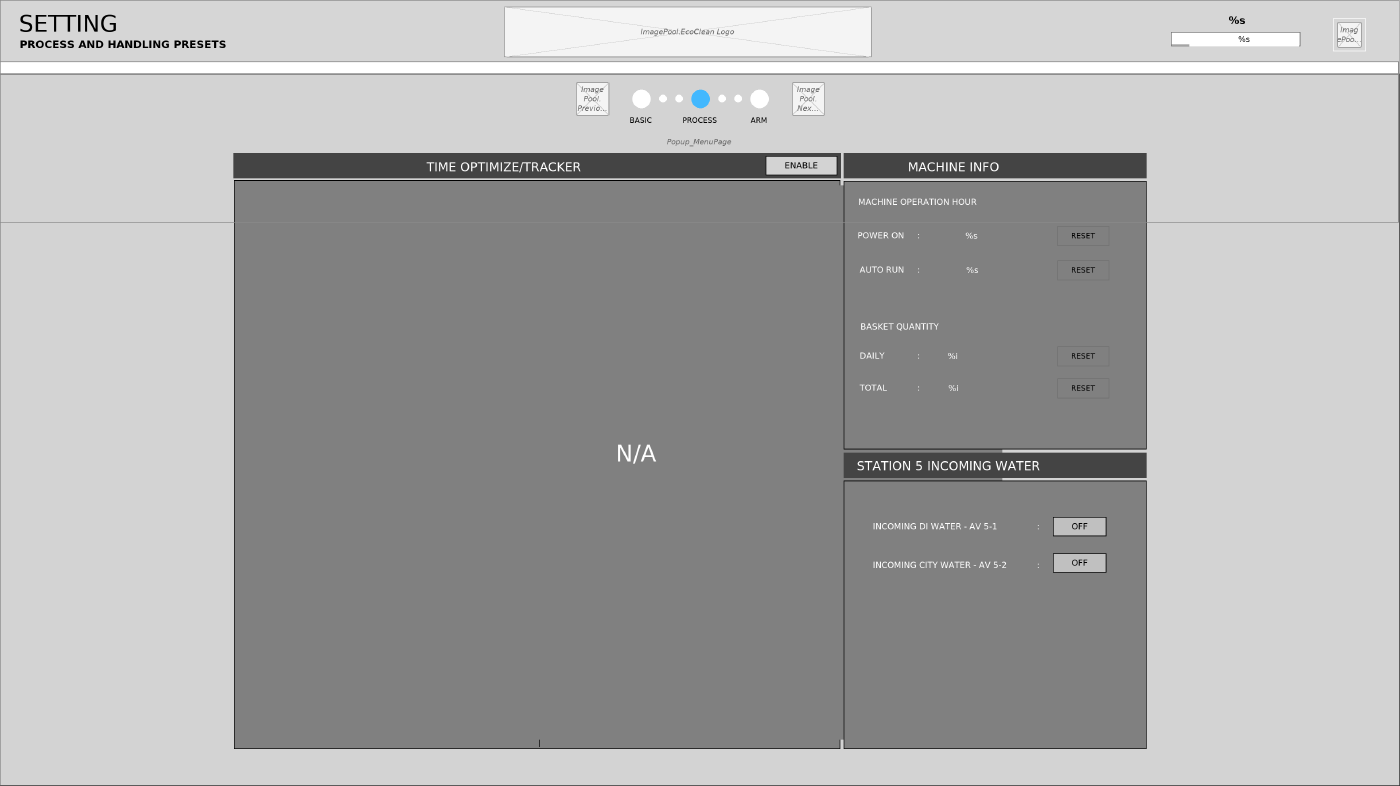
VISUALIZATION SettingProcess_Page  // 1920x1078
    Rectangle (0,101 1920x977)
    Rectangle (321,247 831x780)
    Rectangle (0,63 1920x26)
        p3528305787: HMI_Ctrl.ANIMATION3
    Rectangle (0,0 1919x85)
    Label (23,6 267x53), "SETTING"
    Label (24,49 320x24), "PROCESS AND HANDLING PRESETS"
    Group (1828,25 45x45)
        OnMouseClick: toggle HMI_Ctrl.MenuButton
        RoundedRectangle (0,0 45x45), colour toggle: HMI_Ctrl.MenuButton
        Image (6,5 33x35), image: ImagePool.Menu Button
    Ellipse (867,123 25x25)
    Ellipse (948,123 25x25)
    Ellipse (904,130 10x10)
    Ellipse (926,130 10x10)
    Ellipse (985,130 10x10)
    Ellipse (1007,130 10x10)
    Ellipse (1029,123 25x25)
    Label (847,153 64x24), "BASIC"
    Label (928,153 64x24), "PROCESS"
    Label (1009,153 64x24), "ARM"
    Image (1086,113 45x45), image: ImagePool.Next Button
        OnMouseClick: change screen: SettingArm_Page
    Image (790,113 45x45), image: ImagePool.Previous Button
        OnMouseClick: change screen: Setting_Page
    Rectangle (320,210 833x34)
    Label (582,217 283x24), "TIME OPTIMIZE/TRACKER"
    RoundedRectangle (491,308 30x30), colour toggle: ARbProductRecipeTimeBlockAvailable[1]
    RoundedRectangle (491,378 30x30), colour toggle: ARbProductRecipeTimeBlockAvailable[2]
    RoundedRectangle (491,446 30x30), colour toggle: ARbProductRecipeTimeBlockAvailable[3]
    RoundedRectangle (491,523 30x30), colour toggle: ARbProductRecipeTimeBlockAvailable[4]
    RoundedRectangle (491,598 30x30), colour toggle: ARbProductRecipeTimeBlockAvailable[5]
    RoundedRectangle (491,678 30x30), colour toggle: ARbProductRecipeTimeBlockAvailable[6]
    RoundedRectangle (491,758 30x30), colour toggle: ARbProductRecipeTimeBlockAvailable[7]
    RoundedRectangle (491,829 30x30), colour toggle: ARbProductRecipeTimeBlockAvailable[8]
    RoundedRectangle (491,898 30x30), colour toggle: ARbProductRecipeTimeBlockAvailable[9]
    Label (484,260 103x25), "ENABLE"
    RoundedRectangle (491,968 30x30), colour toggle: ARbProductRecipeTimeBlockAvailable[10]
    Label (385,307 37x24), "1"
    Label (385,377 37x24), "2"
    Label (385,445 37x24), "3"
    Label (385,522 37x24), "4"
    Label (385,597 37x24), "5"
    Label (385,677 37x24), "6"
    Label (385,757 37x24), "7"
    Label (385,828 37x24), "8"
    Label (385,897 37x24), "9"
    Label (380,967 37x24), "10"
    Label (360,248 113x46), "RECIPE NO"
    RoundedRectangle (594,306 90x40), "RESET", input disabled if: bMainOnOff
        tap bTrackerReset[1]
    RoundedRectangle (594,376 90x40), "RESET", input disabled if: bMainOnOff
        tap bTrackerReset[2]
    RoundedRectangle (594,444 90x40), "RESET", input disabled if: bMainOnOff
        tap bTrackerReset[3]
    RoundedRectangle (594,521 90x40), "RESET", input disabled if: bMainOnOff
        tap bTrackerReset[4]
    RoundedRectangle (594,596 90x40), "RESET", input disabled if: bMainOnOff
        tap bTrackerReset[5]
    RoundedRectangle (594,676 90x40), "RESET", input disabled if: bMainOnOff
        tap bTrackerReset[6]
    RoundedRectangle (594,756 90x40), "RESET", input disabled if: bMainOnOff
        tap bTrackerReset[7]
    RoundedRectangle (594,827 90x40), "RESET", input disabled if: bMainOnOff
        tap bTrackerReset[8]
    RoundedRectangle (594,896 90x40), "RESET", input disabled if: bMainOnOff
        tap bTrackerReset[9]
    RoundedRectangle (594,966 90x40), "RESET", input disabled if: bMainOnOff
        tap bTrackerReset[10]
    RoundedRectangle (906,308 30x30), colour toggle: ARbProductRecipeTimeBlockAvailable[11]
    RoundedRectangle (906,378 30x30), colour toggle: ARbProductRecipeTimeBlockAvailable[12]
    RoundedRectangle (906,446 30x30), colour toggle: ARbProductRecipeTimeBlockAvailable[13]
    RoundedRectangle (906,523 30x30), colour toggle: ARbProductRecipeTimeBlockAvailable[14]
    RoundedRectangle (906,598 30x30), colour toggle: ARbProductRecipeTimeBlockAvailable[15]
    RoundedRectangle (906,678 30x30), colour toggle: ARbProductRecipeTimeBlockAvailable[16]
    RoundedRectangle (906,758 30x30), colour toggle: ARbProductRecipeTimeBlockAvailable[17]
    RoundedRectangle (906,829 30x30), colour toggle: ARbProductRecipeTimeBlockAvailable[18]
    RoundedRectangle (906,898 30x30), colour toggle: ARbProductRecipeTimeBlockAvailable[19]
    Label (894,258 103x25), "ENABLE"
    RoundedRectangle (906,968 30x30), colour toggle: ARbProductRecipeTimeBlockAvailable[20]
    Label (803,309 37x24), "11"
    Label (803,379 37x24), "12"
    Label (803,447 37x24), "13"
    Label (803,524 37x24), "14"
    Label (803,599 37x24), "15"
    Label (803,679 37x24), "16"
    Label (803,759 37x24), "17"
    Label (803,830 37x24), "18"
    Label (803,899 37x24), "19"
    Label (802,969 37x24), "20"
    RoundedRectangle (1007,306 90x40), "RESET", input disabled if: bMainOnOff
        tap bTrackerReset[11]
    RoundedRectangle (1007,376 90x40), "RESET", input disabled if: bMainOnOff
        tap bTrackerReset[12]
    RoundedRectangle (1007,444 90x40), "RESET", input disabled if: bMainOnOff
        tap bTrackerReset[13]
    RoundedRectangle (1007,521 90x40), "RESET", input disabled if: bMainOnOff
        tap bTrackerReset[14]
    RoundedRectangle (1007,596 90x40), "RESET", input disabled if: bMainOnOff
        tap bTrackerReset[15]
    RoundedRectangle (1007,676 90x40), "RESET", input disabled if: bMainOnOff
        tap bTrackerReset[16]
    RoundedRectangle (1007,756 90x40), "RESET", input disabled if: bMainOnOff
        tap bTrackerReset[17]
    RoundedRectangle (1007,827 90x40), "RESET", input disabled if: bMainOnOff
        tap bTrackerReset[18]
    RoundedRectangle (1007,896 90x40), "RESET", input disabled if: bMainOnOff
        tap bTrackerReset[19]
    RoundedRectangle (1007,966 90x40), "RESET", input disabled if: bMainOnOff
        tap bTrackerReset[20]
    Label (778,248 113x46), "RECIPE NO"
    Image (691,9 504x69), image: ImagePool.EcoClean Logo
    Rectangle (1050,214 98x26), "ENABLE", colour toggle: bTimeOptimizeDisable, input disabled if: bMainOnOff
        toggle bTimeOptimizeDisable
    Group (1606,17 179x46)
        Button (0,27 177x19), image: VisuSymbols.Symbols.AddUser
        Rectangle (25,28 150x18), "%s", text variable: fbHmiTF1800_UserlevelManagement.dsHmiUserStatus_Active.sLoginName
        Rectangle (2,0 177x22), "%s", text variable: DSLocalSystemTimeML.sCurrentDT24Hr_General
    Line (750,270)
    Line (740,1024) (740,255)
    Group (340,254 783x771), invisible if: bTimeOptimizeDisable
        Rectangle (0,0 1034x760), invisible if: bArmJogEnable
        Label (362,280 341x176), "N/A", invisible if: bArmJogEnable
    Rectangle (1157,248 415x368)
    Rectangle (1157,659 415x368)
    Rectangle (1157,210 415x34)
    Rectangle (1157,621 415x34)
    Label (1242,217 154x24), "MACHINE INFO"
    Label (1174,265 166x24), "MACHINE OPERATION HOUR"
    Label (1173,311 82x24), "POWER ON"
    Label (1176,358 77x24), "AUTO RUN"
    Label (1177,436 134x24), "BASKET QUANTITY"
    Label (1758,515 38x22)
    Rectangle (1248,315 169x17), "%s", text variable: sMachineOnTime_Customer
    Rectangle (1249,362 169x17), "%s", text variable: sMachineRunningTime_Customer
    Label (1176,476 43x24), "DAILY"
    Button (1450,475 71x27), "RESET", colour toggle: bBasketTotalizerResetPB_Daily
        tap bBasketTotalizerResetPB_Daily
    Rectangle (1222,480 169x17), "%i", text variable: diTotalBasketQty_Daily
    Label (1172,627 340x24), "STATION 5 INCOMING WATER"
    Label (1194,710 204x24), "INCOMING DI WATER - AV 5-1"
    Label (1194,763 217x24), "INCOMING CITY WATER - AV 5-2"
    Rectangle (1444,709 73x26), "ON", input disabled if: bMainOnOff
    Rectangle (1444,759 73x26), "ON", input disabled if: bMainOnOff
    Label (1176,520 48x24), "TOTAL"
    Rectangle (1223,524 169x17), "%i", text variable: diTotalBasketQty_Customer
    Button (1450,519 71x27), "RESET", colour toggle: bBasketTotalizerResetPB_Daily
        tap bBasketTotalizerResetPB_User p3779583253=TRUE
    Button (1450,310 71x27), "RESET", colour toggle: bBasketTotalizerResetPB_Daily
        tap bMachineOnTimeRstPB_Customer
    Button (1450,357 71x27), "RESET", colour toggle: bBasketTotalizerResetPB_Daily
        tap bMachineRunningTimeRstPB_Customer
    Rectangle (1444,709 73x26), "OFF", invisible if: ARbOptionSelectedAutoTopupFlag[1], input disabled if: bMainOnOff
        tap ARbOptionSelectedAutoTopupFlag[1]
    Rectangle (1444,759 73x26), "OFF", invisible if: ARbOptionSelectedAutoTopupFlag[2], input disabled if: bMainOnOff
        toggle ARbOptionSelectedAutoTopupFlag[2]
    Label (1255,311 19x24), ":"
    Label (1255,358 19x24), ":"
    Label (1255,476 19x24), ":"
    Label (1255,520 19x24), ":"
    Label (1419,710 19x24), ":"
    Label (1419,763 19x24), ":"
    Frame (0,84 1918x221), invisible if: HMI_Ctrl.CloseMenuButton
        shows Popup_MenuPage()
END_VISUALIZATION

(* stored: Version 1.1.0.1, ProductVersion 3.1.4024.12
   Visu SettingProcess_Page: Id {92b181fa-b85f-41a2-825e-4772c23635fc} *)
